{attribute 'hide_all_locals'}
FUNCTION_BLOCK FB_TcpSendReceiving
VAR_INPUT
	bEnable 			: BOOL; 								//启用
	bReset 				: BOOL; 								//复位,目前设置了自动重连,所以该输入没实现
	sRemoteIp 		: T_IPv4Addr; 						//目标Ip
	nRemotePort 		: UDINT; 								//目标端口
	bExecute 			: BOOL; 								//发送
	pSendData 		: POINTER TO BYTE; 			//发送地址
	nSendSize 		: UDINT; 								//发送数据区域大小
	pRecvData 		: POINTER TO BYTE; 			//接收地址
	nRecvSize 			: UDINT; 								//接收数据区域大小
END_VAR
VAR_OUTPUT
	bBusyConnect 	: BOOL; 								//连接中
	bConnected 		: BOOL; 								//连接完成
	bBusySend 		: BOOL; 								//发送中
	bSendDone 		: BOOL; 								//发送完成
	bBusyRecv 		: BOOL; 								//接受中
	bRecvDone 		: BOOL; 								//接收完成
	bError 				: BOOL; 								//报错
	nRecvBytes 		: UDINT; 								//接收数据长度
	bDataReceived 	: BOOL; 								//接收到数据
END_VAR
VAR
	//功能块调用
	fbConnect : FB_SocketConnect;
	fbClose : FB_SocketClose;
	fbSend : FB_SocketSend;
	fbRecv : FB_SocketReceive;
	
	//状态流转
	stepSendRecv :UDINT;
	stepReceiving : UDINT;
	stepSend : UDINT;
	//连接部分
	tonReconnect : TON;
	hSocket : T_HSOCKET;
	
	//数据收发
	rTrigSend : R_TRIG;
	
	tonRecv : TON;
	tempData : ARRAY[0..MAXBUFFERSIZE] OF BYTE;
	hr: BOOL;
	nCountRecvErr : UDINT;

END_VAR

VAR CONSTANT
	MAXBUFFERSIZE: DINT := 1023;
	EmptyhSocket : T_HSOCKET := (handle := 0);
END_VAR


IF pSendData = 0 OR pRecvData = 0  THEN
	RETURN;
END_IF
//主逻辑
_CyclicLogic();

METHOD PRIVATE _CyclicLogic : BOOL
VAR_INPUT
END_VAR

VAR
END_VAR



tonReconnect(IN:= , PT:= T#3S, Q=> , ET=> );
bBusyConnect := (stepSendRecv <> 20);
bConnected := (stepSendRecv = 20);
bError := fbConnect.bError OR fbClose.bError OR fbSend.bError OR fbRecv.bError;

CASE stepSendRecv OF
	0: //初始状态，等待TCP连接
	fbConnect(bExecute:= FALSE);
	fbClose(bExecute:= FALSE);
	fbSend(bExecute:= FALSE);
	fbRecv(bExecute := FALSE);
	tonReconnect.IN := FALSE;
	nCountRecvErr := 0;
	IF bEnable AND sRemoteIp <> '' AND nRemotePort <> 0 THEN
		stepSendRecv := 10;
	END_IF

	10: //连接中
	fbConnect(sRemoteHost:= sRemoteIp, nRemotePort:= nRemotePort, bExecute:= TRUE);
	IF fbConnect.bBusy THEN
		;
	ELSE
		IF NOT fbConnect.bError AND (fbConnect.hSocket.handle <> 0) THEN
			hSocket := fbConnect.hSocket;
			stepSendRecv := 20;
		ELSE
			stepSendRecv := 12;
		END_IF
	END_IF

	12: //重连等待
	tonReconnect.IN := TRUE;
	IF tonReconnect.Q THEN
		stepSendRecv := 0;
		tonReconnect.IN := FALSE;
	END_IF

	20: //连接完成
	_Send();
	hr := _Receiving(200,6);
	IF hr = TRUE THEN
		stepSendRecv := 30;
	END_IF
	
	
	30:
	fbClose(hSocket:= hSocket, bExecute:= TRUE );
	IF fbClose.bBusy THEN
		;
	ELSE
		hSocket := EmptyhSocket;
		stepSendRecv := 0;
	END_IF
END_CASE
END_METHOD

METHOD PRIVATE _Receiving : BOOL
VAR_INPUT
	CycleTime : UDINT;
	ErrorLimit : UDINT;
END_VAR
tonRecv(IN:= , PT:= UDINT_TO_TIME(CycleTime), Q=> , ET=> );
bBusyRecv := (stepReceiving = 10 );
bRecvDone := (stepReceiving <> 10 );
CASE stepReceiving OF
	0:
	bDataReceived := FALSE;
	tonRecv.IN := FALSE;
	fbRecv(bExecute := FALSE);
	stepReceiving := 10;
	
	10:
	
	fbRecv(hSocket:= hSocket, cbLen:= SIZEOF(tempData), pDest:= ADR(tempData), bExecute:= TRUE);
	IF fbRecv.bBusy THEN
		;
	ELSE
		IF fbRecv.bError THEN
			nCountRecvErr := nCountRecvErr + 1;
			_Receiving := (nCountRecvErr > ErrorLimit);
		ELSE
			nCountRecvErr := 0;
			IF fbRecv.nRecBytes <> 0 THEN
				MEMSET(destAddr:= pRecvData, fillByte:= 0, n:= nRecvSize);
				MEMCPY(destAddr:= pRecvData, srcAddr:= ADR(tempData), n:= MIN(fbRecv.nRecBytes,nRecvSize) );
				bDataReceived := TRUE;
			END_IF
			nRecvBytes := fbRecv.nRecBytes;
		END_IF
		stepReceiving := 20;
		tonRecv.IN := TRUE;
	END_IF

	20:
	
	tonRecv.IN := TRUE;
	IF tonRecv.Q THEN
		tonRecv.IN := FALSE;
		stepReceiving := 0;
	END_IF

END_CASE
END_METHOD

METHOD PRIVATE _Send : BOOL
VAR_INPUT
END_VAR
rTrigSend(CLK:= bExecute, Q=> );
bBusySend := (stepSend <> 0);
bSendDone := (stepSend = 0);
CASE stepSend OF
	0:
	fbSend(bExecute:= FALSE);
	IF rTrigSend.Q THEN
		stepSend := 10;

	END_IF
	
	
	10:
	fbSend(hSocket:= hSocket, cbLen:= nSendSize, pSrc:= pSendData, bExecute:= TRUE);
	IF fbSend.bBusy THEN
		;
	ELSE
		IF fbSend.bError THEN
			_Send := TRUE;
		ELSE
			;
		END_IF
		stepSend := 0;
	END_IF
	

END_CASE
END_METHOD

END_FUNCTION_BLOCK

(* stored: Version 1.1.0.1, ProductVersion 3.1.4024.12
   POU FB_TcpSendReceiving: Id {11aa6855-73f2-4b06-a2d2-8a40a5343dc1}, SpecialFunc None
   Method _CyclicLogic: Id {69b2bd2c-1ad8-42d5-a8f8-6209c3df6db1}
   Method _Receiving: Id {41a25567-f4c4-4515-a635-213bf395acab}
   Method _Send: Id {a364897d-e130-4944-9ef2-507dffe27e1c} *)
